TYPE ControlBESScmds :
STRUCT
	start: BOOL;
END_STRUCT
END_TYPE

(* stored: Version 1.1.0.1, ProductVersion 3.1.4024.4
   DUT ControlBESScmds: Id {a4c29788-5bc5-4651-917c-6aee35987d05} *)
